TYPE OutputBase_10CEE7DE :
STRUCT
END_STRUCT
END_TYPE

(* stored: Version 1.2.0.0, ProductVersion 3.1.4024.11
   DUT OutputBase_10CEE7DE: Id {bbabb1dd-04cb-4f04-8190-dbfc188de32a} *)
